KUKA KRL data list: Glode_HanGao.dat

&ACCESS RVO1
&REL 298
&PARAM EDITMASK = *
&PARAM TEMPLATE = C:\KRC\Roboter\Template\vorgabe
&PARAM DISKPATH = KRC:\R1\Program\HK
DEFDAT  glode_hangao PUBLIC




;--------DECL_Enum---------------
GLOBAL ENUM Sink_Type_Enum UpDown_One,LeftRight_One,LeftRight_Two,Null
GLOBAL ENUM Area_Enum L0,C45,L90,C135,L180,C225,L270,C315,N45,N135,N225,N315
GLOBAL ENUM Pos_Type_Enum C_LIN_POS,C_CIR_POS,L_LIN_POS
GLOBAL ENUM Work_Area_Enum A0,A90,A270
GLOBAL ENUM Vision_Model_Enum Calibration,Find_Model
;----------------------------------
;---DECL-STRUC-------------------------


GLOBAL STRUC Surround_Welding_Type BOOL Write_Status,REAL Sink_Size_Long,REAL Sink_Size_Width,REAL Sink_Size_R,REAL Sink_Size_Short_Side,REAL Sink_Size_Short_OnePos,REAL Sink_Size_Short_TwoPos,REAL Sink_Size_Pots_Thick,REAL Sink_Size_Panel_Thick,INT Sink_Model,REAL Sink_Size_Left_Distance,REAL Sink_Size_Down_Distance,Sink_Type_Enum Sink_Type
GLOBAL STRUC LSC_TOOL_TYP INT LSR_MAX_PWR,INT LSR_MIN_PWR,INT LSR_Prg,REAL SNSR_Prg,INT SNSR_State,REAL GAS_Pressure,INT LSR_Dly,INT GAS_Pre_Flow,INT GAS_Post_Flow
GLOBAL STRUC Offset_POS REAL X,REAL Y,REAL Z,REAL A,REAL B,REAL C
GLOBAL STRUC Offset_CIR REAL C_X,REAL C_Y,REAL C_Z,REAL C_A,REAL C_B,REAL C_C
GLOBAL STRUC Calculate_Lin_Const REAL A,REAL B,REAL C
GLOBAL STRUC Calibration_Sink_TYP REAL Long,REAL Width




GLOBAL STRUC Surr_Welding_Craft_Type CHAR Welding_Name[20],E6POS Welding_Pos,REAL Welding_Power,REAL Welding_Speed,REAL Welding_Angle,INT Welding_CDIS,INT Welding_ACC,Offset_POS Welding_Offset,Offset_CIR Welding_Offset_CIR





;-------------------------------------


;----------DECL_Value----------------------
DECL GLOBAL Surround_Welding_Type SW_DEFAULT={Sink_Size_Long 50.0000,Sink_Size_Width 345.000,Sink_Size_R 10.0000,Sink_Size_Pots_Thick 0.750000,Sink_Size_Panel_Thick 2.85000,Sink_Model 952154,Sink_Type #UpDown_One}
DECL GLOBAL LSC_TOOL_TYP LTDEFAULT={LSR_MAX_PWR 500,LSR_MIN_PWR 50,LSR_Prg 1,SNSR_Prg 1.00000,SNSR_State 0,GAS_Pressure 1.00000,LSR_Dly 100,GAS_Pre_Flow 0,GAS_Post_Flow 0}
DECL GLOBAL Offset_POS FFDEFAULT={X 0.0,Y 0.0,Z 0.0,A 0.0,B 0.0,C 0.0}
DECL GLOBAL Offset_CIR FCDEFAULT={C_X 0.0,C_Y 0.0,C_Z 0.0,C_A 0.0,C_B 0.0,C_C 0.0}
DECL GLOBAL E6POS PODEFAULT={X 0.0,Y 0.0,Z 0.0,A 0.0,B 0.0,C 0.0}


DECL GLOBAL Surround_Welding_Type Camera_Calibration_Data={Sink_Size_Long 632.000,Sink_Size_Width 352.000,Sink_Size_R 10.0000,Sink_Size_Short_Side 23.0000,Sink_Size_Short_OnePos 36.0000,Sink_Size_Short_TwoPos 328.000,Sink_Size_Pots_Thick 0.750000,Sink_Size_Panel_Thick 0.0,Sink_Model 952154,Sink_Size_Left_Distance 24.0000,Sink_Size_Down_Distance 24.0000,Sink_Type #LeftRight_One}

DECL GLOBAL E6POS N1_Cam_45_POS={X 1765.00,Y -1.00106740E-34,Z 1784.00,A 0.0,B 90.0000,C 3.24968513E-36}
DECL GLOBAL E6POS N1_Cam_135_POS={X 1765.00,Y -9.34353299E-23,Z 1784.00,A 0.0,B 90.0000,C 3.03311614E-24}
DECL GLOBAL E6POS N1_Cam_225_POS={X 1765.00,Y 5.47478833E-11,Z 1784.00,A 0.0,B 90.0000,C -6.59667199E-13}
DECL GLOBAL E6POS N1_Cam_315_POS={X 0.0,Y 0.0,A 0.0,B 0.0,C 0.0}

DECL GLOBAL E6POS N2_Cam_45_POS={X 293.122131,Y 89.9176636,Z -80.0293961,A 0.441927105,B -0.0416148715,C -0.0704164580,S 'B0010',T 'B1010',E1 0.0,E2 0.0,E3 0.0,E4 0.0,E5 0.0,E6 0.0}
DECL GLOBAL E6POS N2_Cam_135_POS={X -42.3839874,Y 91.8151550,Z -80.0254822,A 0.441927105,B -0.0416148864,C -0.0704164430,S 'B0010',T 'B1010',E1 0.0,E2 0.0,E3 0.0,E4 0.0,E5 0.0,E6 0.0}
DECL GLOBAL E6POS N2_Cam_225_POS={X -39.7999954,Y 716.082336,Z -80.0293350,A 0.441926539,B -0.0416153781,C -0.0704161152,S 'B0010',T 'B00101011',E1 0.0,E2 0.0,E3 0.0,E4 0.0,E5 0.0,E6 0.0}
DECL GLOBAL E6POS N2_Cam_315_POS={X 294.984924,Y 714.198059,Z -80.0293350,A 0.441925645,B -0.0416159667,C -0.0704158247,S 'B0010',T 'B00101011',E1 0.0,E2 0.0,E3 0.0,E4 0.0,E5 0.0,E6 0.0}

DECL GLOBAL E6POS N45_OFFSET_POS={X 375.675,Y 23.4770,Z 0.0,A 0.0,B 0.0,C 0.0}
DECL GLOBAL E6POS N135_OFFSET_POS={X 24.0190,Y 23.1910,Z 0.0,A 0.0,B 0.0,C 0.0}
DECL GLOBAL E6POS N225_OFFSET_POS={X 23.4020,Y 725.222,Z 0.0,A 0.0,B 0.0,C 0.0}
DECL GLOBAL E6POS N315_OFFSET_POS={X 375.730,Y 725.747,Z 0.0,A 0.0,B 0.0,C 0.0}

DECL GLOBAL E6POS N45_CIR_POS={X 372.590,Y 27.2660,Z 0.0,A 0.0,B 0.0,C 0.0}
DECL GLOBAL E6POS N135_CIR_POS={X 27.7730,Y 26.2530,Z 0.0,A 0.0,B 0.0,C 0.0}
DECL GLOBAL E6POS N225_CIR_POS={X 27.3020,Y 722.048,Z 0.0,A 0.0,B 0.0,C 0.0}
DECL GLOBAL E6POS N315_CIR_POS={X 372.023,Y 722.369,Z 0.0,A 0.0,B 0.0,C 0.0}

DECL GLOBAL E6POS D45_Start_POS={X 364.343,Y -0.734000,Z 0.0,A 0.0,B 0.0,C 0.0}
DECL GLOBAL E6POS D45_End_POS={X 364.315,Y 23.5880,Z 0.0,A 0.0,B 0.0,C 0.0}
DECL GLOBAL E6POS D135_Start_POS={X 37.1160,Y -1.02700,Z 0.0,A 0.0,B 0.0,C 0.0}
DECL GLOBAL E6POS D135_End_POS={X 37.2780,Y 23.2150,Z 0.0,A 0.0,B 0.0,C 0.0}
DECL GLOBAL E6POS D225_Start_POS={X 36.7810,Y 749.275,Z 0.0,A 0.0,B 0.0,C 0.0}
DECL GLOBAL E6POS D225_End_POS={X 36.9310,Y 725.260,Z 0.0,A 0.0,B 0.0,C 0.0}
DECL GLOBAL E6POS D315_Start_POS={X 364.063,Y 750.089,Z 0.0,A 0.0,B 0.0,C 0.0}
DECL GLOBAL E6POS D315_End_POS={X 364.380,Y 725.694,Z 0.0,A 0.0,B 0.0,C 0.0}


DECL GLOBAL Surr_Welding_Craft_Type L0_Welding_Craft[2,10]
L0_Welding_Craft[1,1]={Welding_Name[] "S2",Welding_Pos {X 120.000,Y 38.0000,Z 0.0,A 0.0,B 20.0000,C 0.0},Welding_Power 80.0000,Welding_Speed 0.0400000,Welding_Angle 20.0000,Welding_CDIS 5,Welding_ACC 100,Welding_Offset {X 0.0,Y 0.0,Z 0.0}}
L0_Welding_Craft[1,2]={Welding_Name[] "L0_S2",Welding_Pos {X 376.000,Y 584.800,Z 0.0,A 0.0,B 20.0000,C 0.0},Welding_Power 80.0000,Welding_Speed 0.0400000,Welding_Angle 20.0000,Welding_CDIS 5,Welding_ACC 100,Welding_Offset {X 0.0,Y 0.0,Z 0.0}}
L0_Welding_Craft[1,3]={Welding_Name[] "L0_S3",Welding_Pos {X 376.000,Y 340.000,Z 0.0,A 0.0,B 20.0000,C 0.0},Welding_Power 80.0000,Welding_Speed 0.0400000,Welding_Angle 20.0000,Welding_CDIS 5,Welding_ACC 100,Welding_Offset {X 0.0,Y 0.0,Z 0.0}}
L0_Welding_Craft[1,4]={Welding_Name[] "L0_S4",Welding_Pos {X 376.000,Y 64.6000061,Z 0.0,A 0.0,B 20.0000,C 0.0},Welding_Power 80.0000,Welding_Speed 0.0400000,Welding_Angle 20.0000,Welding_CDIS 5,Welding_ACC 100,Welding_Offset {X 0.0,Y 0.0,Z 0.0}}
L0_Welding_Craft[1,5]={Welding_Name[] "S1",Welding_Pos {X 400.000,Y 86.0000153,Z -3.00000,A 0.0,B 23.0000,C 0.0},Welding_Power 80.0000,Welding_Speed 0.0400000,Welding_Angle 20.0000,Welding_CDIS 5,Welding_ACC 100,Welding_Offset {X 0.0,Y 0.0,Z 0.0}}
L0_Welding_Craft[1,6]={Welding_Name[] "S6",Welding_Pos {X 533.000,Y 463.600037,Z -2.05000,A 0.0,B -23.0000,C 0.0},Welding_Power 80.0000,Welding_Speed 0.0400000,Welding_Angle 20.0000,Welding_CDIS 5,Welding_ACC 100,Welding_Offset {X 0.0,Y 0.0,Z 0.0}}
L0_Welding_Craft[1,7]={Welding_Name[] "S7",Welding_Pos {X 533.000,Y 463.600037,Z -2.05000,A 0.0,B -23.0000,C 0.0},Welding_Power 80.0000,Welding_Speed 0.0400000,Welding_Angle 20.0000,Welding_CDIS 5,Welding_ACC 100,Welding_Offset {X 0.0,Y 0.0,Z 0.0}}
L0_Welding_Craft[1,8]={Welding_Name[] "S8",Welding_Pos {X 533.000,Y 463.600037,Z -2.05000,A 0.0,B -23.0000,C 0.0},Welding_Power 80.0000,Welding_Speed 0.0400000,Welding_Angle 20.0000,Welding_CDIS 5,Welding_ACC 100,Welding_Offset {X 0.0,Y 0.0,Z 0.0}}
L0_Welding_Craft[1,9]={Welding_Name[] "S9",Welding_Pos {X 533.000,Y 463.600037,Z -2.05000,A 0.0,B -23.0000,C 0.0},Welding_Power 80.0000,Welding_Speed 0.0400000,Welding_Angle 20.0000,Welding_CDIS 5,Welding_ACC 100,Welding_Offset {X 0.0,Y 0.0,Z 0.0}}
L0_Welding_Craft[1,10]={Welding_Name[] "S10",Welding_Pos {X 533.000,Y 338.000,Z -2.05000,A 0.0,B -23.0000,C 0.0},Welding_Power 80.0000,Welding_Speed 0.0400000,Welding_Angle 20.0000,Welding_CDIS 5,Welding_ACC 100,Welding_Offset {X 0.0,Y 0.0,Z 0.0}}
L0_Welding_Craft[2,1]={Welding_Name[] "L0_S1",Welding_Pos {X 375.681122,Y 101.703979,Z 0.0,A 0.0,B 20.0000,C 0.0},Welding_Power 80.0000,Welding_Speed 0.300000,Welding_Angle 20.0000,Welding_CDIS 5,Welding_ACC 100,Welding_Offset {X 0.0,Y 0.0,Z 0.0}}
L0_Welding_Craft[2,2]={Welding_Name[] "L0_S2",Welding_Pos {X 375.566071,Y 647.351257,Z 0.0,A 0.0,B 20.0000,C 0.0},Welding_Power 80.0000,Welding_Speed 0.0320000,Welding_Angle 20.0000,Welding_CDIS 5,Welding_ACC 100,Welding_Offset {X 0.0,Y -1.50000,Z 0.0}}
L0_Welding_Craft[2,3]={Welding_Name[] "L0_S3",Welding_Pos {X 375.650,Y 374.428497,Z 0.0,A 0.0,B 20.0000,C 0.0},Welding_Power 80.0000,Welding_Speed 0.0320000,Welding_Angle 20.0000,Welding_CDIS 5,Welding_ACC 100,Welding_Offset {X 0.0,Y -1.80000,Z 0.0}}
L0_Welding_Craft[2,4]={Welding_Name[] "L0_S4",Welding_Pos {X 375.744415,Y 67.3903809,Z 0.0,A 0.0,B 20.0000,C 0.0},Welding_Power 80.0000,Welding_Speed 0.0340000,Welding_Angle 20.0000,Welding_CDIS 5,Welding_ACC 100,Welding_Offset {X 0.0,Y -1.00000,Z 0.0}}
L0_Welding_Craft[2,5]={Welding_Name[] "S1",Welding_Pos {X 400.000,Y 86.0000153,Z -3.00000,A 0.0,B 23.0000,C 0.0},Welding_Power 80.0000,Welding_Speed 0.0400000,Welding_Angle 20.0000,Welding_CDIS 5,Welding_ACC 100,Welding_Offset {X 0.0,Y 0.0,Z 0.0}}
L0_Welding_Craft[2,6]={Welding_Name[] "S6",Welding_Pos {X 533.000,Y 463.600037,Z -2.05000,A 0.0,B -23.0000,C 0.0},Welding_Power 80.0000,Welding_Speed 0.0400000,Welding_Angle 20.0000,Welding_CDIS 5,Welding_ACC 100,Welding_Offset {X 0.0,Y 0.0,Z 0.0}}
L0_Welding_Craft[2,7]={Welding_Name[] "S7",Welding_Pos {X 533.000,Y 463.600037,Z -2.05000,A 0.0,B -23.0000,C 0.0},Welding_Power 80.0000,Welding_Speed 0.0400000,Welding_Angle 20.0000,Welding_CDIS 5,Welding_ACC 100,Welding_Offset {X 0.0,Y 0.0,Z 0.0}}
L0_Welding_Craft[2,8]={Welding_Name[] "S8",Welding_Pos {X 533.000,Y 463.600037,Z -2.05000,A 0.0,B -23.0000,C 0.0},Welding_Power 80.0000,Welding_Speed 0.0400000,Welding_Angle 20.0000,Welding_CDIS 5,Welding_ACC 100,Welding_Offset {X 0.0,Y 0.0,Z 0.0}}
L0_Welding_Craft[2,9]={Welding_Name[] "S9",Welding_Pos {X 533.000,Y 463.600037,Z -2.05000,A 0.0,B -23.0000,C 0.0},Welding_Power 80.0000,Welding_Speed 0.0400000,Welding_Angle 20.0000,Welding_CDIS 5,Welding_ACC 100,Welding_Offset {X 0.0,Y 0.0,Z 0.0}}
L0_Welding_Craft[2,10]={Welding_Name[] "S10",Welding_Pos {X 533.000,Y 338.000,Z -2.05000,A 0.0,B -23.0000,C 0.0},Welding_Power 80.0000,Welding_Speed 0.0400000,Welding_Angle 20.0000,Welding_CDIS 5,Welding_ACC 100,Welding_Offset {X 0.0,Y 0.0,Z 0.0}}



DECL GLOBAL Surr_Welding_Craft_Type C45_Welding_Craft[2,3]
C45_Welding_Craft[1,1]={Welding_Name[] "S3",Welding_Pos {X 120.000,Y 30.0000,Z 0.0,A 0.0,B 20.0000,C 0.0},Welding_Power 80.0000,Welding_Speed 0.0400000,Welding_Angle 20.0000,Welding_CDIS 5,Welding_ACC 100,Welding_Offset {X 0.0,Y 0.0,Z 0.0}}
C45_Welding_Craft[1,2]={Welding_Name[] "PM2",Welding_Pos {X 117.070,Y 22.9300,Z 0.0,A 0.0,B 0.0,C 0.0},Welding_Power 80.0000,Welding_Speed 0.0400000,Welding_Angle 20.0000,Welding_CDIS 5,Welding_ACC 100,Welding_Offset {X 0.0,Y 0.0,Z 0.0},Welding_Offset_CIR {C_X 0.0,C_Y 0.0,C_Z 0.0}}
C45_Welding_Craft[1,3]={Welding_Name[] "PE2",Welding_Pos {X 110.000,Y 20.0000,Z 0.0,A 0.0,B 0.0,C 20.0000},Welding_Power 80.0000,Welding_Speed 0.0400000,Welding_Angle 20.0000,Welding_CDIS 5,Welding_ACC 100,Welding_Offset {X 0.0,Y 0.0,Z 0.0}}
C45_Welding_Craft[2,1]={Welding_Name[] "C45_S1",Welding_Pos {X 375.754913,Y 33.2750244,Z 0.0,A 0.0,B 20.0000,C 0.0},Welding_Power 80.0000,Welding_Speed 0.0300000,Welding_Angle 20.0000,Welding_CDIS 5,Welding_ACC 100,Welding_Offset {X 0.0,Y 0.0,Z 0.0}}
C45_Welding_Craft[2,2]={Welding_Name[] "PM3",Welding_Pos {X 372.649,Y 27.0560,Z 0.0,A 0.0,B 0.0,C 0.0},Welding_Power 80.0000,Welding_Speed 0.0400000,Welding_Angle 20.0000,Welding_CDIS 5,Welding_ACC 100,Welding_Offset {X 0.0,Y 0.500000,Z 0.0},Welding_Offset_CIR {C_X 0.0,C_Y 0.0,C_Z 0.0}}
C45_Welding_Craft[2,3]={Welding_Name[] "PE3",Welding_Pos {X 365.758,Y 23.2745743,Z 0.0,A 0.0,B 0.0,C 20.0000},Welding_Power 80.0000,Welding_Speed 0.0120000,Welding_Angle 20.0000,Welding_CDIS 5,Welding_ACC 100,Welding_Offset {X 0.0,Y 0.500000,Z 0.0}}


DECL GLOBAL Surr_Welding_Craft_Type L90_Welding_Craft[2,10]
L90_Welding_Craft[1,1]={Welding_Name[] "S2",Welding_Pos {X 30.0000,Y 20.0000,Z 0.0,A 0.0,B 0.0,C 20.0000},Welding_Power 80.0000,Welding_Speed 0.0400000,Welding_Angle 20.0000,Welding_CDIS 5,Welding_ACC 100,Welding_Offset {X 0.0,Y 0.0,Z 0.0}}
L90_Welding_Craft[1,2]={Welding_Name[] "L90_S2",Welding_Pos {X 200.000,Y 24.0000,Z 0.0,A 0.0,B 0.0,C 20.0000},Welding_Power 80.0000,Welding_Speed 0.0400000,Welding_Angle 20.0000,Welding_CDIS 5,Welding_ACC 100,Welding_Offset {X 0.0,Y 0.0,Z 0.0}}
L90_Welding_Craft[1,3]={Welding_Name[] "L90_S3",Welding_Pos {X 67.2000122,Y 24.0000,Z 0.0,A 0.0,B 0.0,C 20.0000},Welding_Power 80.0000,Welding_Speed 0.0400000,Welding_Angle 20.0000,Welding_CDIS 5,Welding_ACC 100,Welding_Offset {X 0.0,Y 0.0,Z 0.0}}
L90_Welding_Craft[1,4]={Welding_Name[] "S4",Welding_Pos {X 400.000,Y 86.0000153,Z -3.00000,A 0.0,B 23.0000,C 0.0},Welding_Power 80.0000,Welding_Speed 0.0400000,Welding_Angle 20.0000,Welding_CDIS 5,Welding_ACC 100,Welding_Offset {X 0.0,Y 0.0,Z 0.0}}
L90_Welding_Craft[1,5]={Welding_Name[] "S5",Welding_Pos {X 371.000,Y 0.0,Z -3.00000,A 0.0,B 0.0,C 23.0000},Welding_Power 80.0000,Welding_Speed 0.0400000,Welding_Angle 20.0000,Welding_CDIS 5,Welding_ACC 100,Welding_Offset {X 0.0,Y 0.0,Z 0.0}}
L90_Welding_Craft[1,6]={Welding_Name[] "S6",Welding_Pos {X 533.000,Y 463.600037,Z -2.05000,A 0.0,B -23.0000,C 0.0},Welding_Power 80.0000,Welding_Speed 0.0400000,Welding_Angle 20.0000,Welding_CDIS 5,Welding_ACC 100,Welding_Offset {X 0.0,Y 0.0,Z 0.0}}
L90_Welding_Craft[1,7]={Welding_Name[] "S7",Welding_Pos {X 533.000,Y 463.600037,Z -2.05000,A 0.0,B -23.0000,C 0.0},Welding_Power 80.0000,Welding_Speed 0.0400000,Welding_Angle 20.0000,Welding_CDIS 5,Welding_ACC 100,Welding_Offset {X 0.0,Y 0.0,Z 0.0}}
L90_Welding_Craft[1,8]={Welding_Name[] "S8",Welding_Pos {X 533.000,Y 463.600037,Z -2.05000,A 0.0,B -23.0000,C 0.0},Welding_Power 80.0000,Welding_Speed 0.0400000,Welding_Angle 20.0000,Welding_CDIS 5,Welding_ACC 100,Welding_Offset {X 0.0,Y 0.0,Z 0.0}}
L90_Welding_Craft[1,9]={Welding_Name[] "S9",Welding_Pos {X 533.000,Y 463.600037,Z -2.05000,A 0.0,B -23.0000,C 0.0},Welding_Power 80.0000,Welding_Speed 0.0400000,Welding_Angle 20.0000,Welding_CDIS 5,Welding_ACC 100,Welding_Offset {X 0.0,Y 0.0,Z 0.0}}
L90_Welding_Craft[1,10]={Welding_Name[] "S10",Welding_Pos {X 533.000,Y 338.000,Z -2.05000,A 0.0,B -23.0000,C 0.0},Welding_Power 80.0000,Welding_Speed 0.0400000,Welding_Angle 20.0000,Welding_CDIS 5,Welding_ACC 100,Welding_Offset {X 0.0,Y 0.0,Z 0.0}}
L90_Welding_Craft[2,1]={Welding_Name[] "L90_S1",Welding_Pos {X 332.548584,Y 23.2731590,Z 0.0,A 0.0,B 0.0,C 20.0000},Welding_Power 80.0000,Welding_Speed 0.0320000,Welding_Angle 20.0000,Welding_CDIS 5,Welding_ACC 100,Welding_Offset {X 0.0,Y 0.800000,Z 0.0}}
L90_Welding_Craft[2,2]={Welding_Name[] "L90_S2",Welding_Pos {X 199.711,Y 23.2675,Z 0.0,A 0.0,B 0.0,C 20.0000},Welding_Power 80.0000,Welding_Speed 0.0320000,Welding_Angle 20.0000,Welding_CDIS 5,Welding_ACC 100,Welding_Offset {X 0.0,Y 0.800000,Z 0.0}}
L90_Welding_Craft[2,3]={Welding_Name[] "L90_S3",Welding_Pos {X 66.8734131,Y 23.2618408,Z 0.0,A 0.0,B 0.0,C 20.0000},Welding_Power 80.0000,Welding_Speed 0.0320000,Welding_Angle 20.0000,Welding_CDIS 5,Welding_ACC 100,Welding_Offset {X 0.0,Y 0.800000,Z 0.0}}
L90_Welding_Craft[2,4]={Welding_Name[] "S4",Welding_Pos {X 400.000,Y 86.0000153,Z -3.00000,A 0.0,B 23.0000,C 0.0},Welding_Power 80.0000,Welding_Speed 0.0400000,Welding_Angle 20.0000,Welding_CDIS 5,Welding_ACC 100,Welding_Offset {X 0.0,Y 0.0,Z 0.0}}
L90_Welding_Craft[2,5]={Welding_Name[] "S5",Welding_Pos {X 371.000,Y 0.0,Z -3.00000,A 0.0,B 0.0,C 23.0000},Welding_Power 80.0000,Welding_Speed 0.0400000,Welding_Angle 20.0000,Welding_CDIS 5,Welding_ACC 100,Welding_Offset {X 0.0,Y 0.0,Z 0.0}}
L90_Welding_Craft[2,6]={Welding_Name[] "S6",Welding_Pos {X 533.000,Y 463.600037,Z -2.05000,A 0.0,B -23.0000,C 0.0},Welding_Power 80.0000,Welding_Speed 0.0400000,Welding_Angle 20.0000,Welding_CDIS 5,Welding_ACC 100,Welding_Offset {X 0.0,Y 0.0,Z 0.0}}
L90_Welding_Craft[2,7]={Welding_Name[] "S7",Welding_Pos {X 533.000,Y 463.600037,Z -2.05000,A 0.0,B -23.0000,C 0.0},Welding_Power 80.0000,Welding_Speed 0.0400000,Welding_Angle 20.0000,Welding_CDIS 5,Welding_ACC 100,Welding_Offset {X 0.0,Y 0.0,Z 0.0}}
L90_Welding_Craft[2,8]={Welding_Name[] "S8",Welding_Pos {X 533.000,Y 463.600037,Z -2.05000,A 0.0,B -23.0000,C 0.0},Welding_Power 80.0000,Welding_Speed 0.0400000,Welding_Angle 20.0000,Welding_CDIS 5,Welding_ACC 100,Welding_Offset {X 0.0,Y 0.0,Z 0.0}}
L90_Welding_Craft[2,9]={Welding_Name[] "S9",Welding_Pos {X 533.000,Y 463.600037,Z -2.05000,A 0.0,B -23.0000,C 0.0},Welding_Power 80.0000,Welding_Speed 0.0400000,Welding_Angle 20.0000,Welding_CDIS 5,Welding_ACC 100,Welding_Offset {X 0.0,Y 0.0,Z 0.0}}
L90_Welding_Craft[2,10]={Welding_Name[] "S10",Welding_Pos {X 533.000,Y 338.000,Z -2.05000,A 0.0,B -23.0000,C 0.0},Welding_Power 80.0000,Welding_Speed 0.0400000,Welding_Angle 20.0000,Welding_CDIS 5,Welding_ACC 100,Welding_Offset {X 0.0,Y 0.0,Z 0.0}}

DECL GLOBAL Surr_Welding_Craft_Type C135_Welding_Craft[2,3]
C135_Welding_Craft[1,1]={Welding_Name[] "S3",Welding_Pos {X 30.0000,Y 20.0000,Z 0.0,A 0.0,B 0.0,C 20.0000},Welding_Power 80.0000,Welding_Speed 0.0400000,Welding_Angle 20.0000,Welding_CDIS 5,Welding_ACC 100,Welding_Offset {X 0.0,Y 0.0,Z 0.0}}
C135_Welding_Craft[1,2]={Welding_Name[] "PM3",Welding_Pos {X 22.9300,Y 22.9300,Z 0.0,A 0.0,B 0.0,C 0.0},Welding_Power 80.0000,Welding_Speed 0.0400000,Welding_Angle -20.0000,Welding_CDIS 5,Welding_ACC 100,Welding_Offset {X 0.0,Y 0.0,Z 0.0},Welding_Offset_CIR {C_X 0.0,C_Y 0.0,C_Z 0.0}}
C135_Welding_Craft[1,3]={Welding_Name[] "PE3",Welding_Pos {X 20.0000,Y 30.0000,Z 0.0,A 0.0,B -20.0000,C 0.0},Welding_Power 80.0000,Welding_Speed 0.0400000,Welding_Angle -20.0000,Welding_CDIS 5,Welding_ACC 100,Welding_Offset {X 0.0,Y 0.0,Z 0.0}}
C135_Welding_Craft[2,1]={Welding_Name[] "C135_S1",Welding_Pos {X 33.6640,Y 23.2604256,Z 0.0,A 0.0,B 0.0,C 20.0000},Welding_Power 80.0000,Welding_Speed 0.0300000,Welding_Angle 20.0000,Welding_CDIS 5,Welding_ACC 100,Welding_Offset {X 0.0,Y 0.500000,Z 0.0}}
C135_Welding_Craft[2,2]={Welding_Name[] "PM4",Welding_Pos {X 27.4390,Y 26.3430,Z 0.0,A 0.0,B 0.0,C 0.0},Welding_Power 80.0000,Welding_Speed 0.0400000,Welding_Angle -20.0000,Welding_CDIS 5,Welding_ACC 100,Welding_Offset {X 0.0,Y 0.0,Z 0.0},Welding_Offset_CIR {C_X 0.0,C_Y 0.0,C_Z 0.0}}
C135_Welding_Craft[2,3]={Welding_Name[] "PE4",Welding_Pos {X 23.6575489,Y 33.2600,Z 0.0,A 0.0,B -20.0000,C 0.0},Welding_Power 80.0000,Welding_Speed 0.0150000,Welding_Angle -20.0000,Welding_CDIS 5,Welding_ACC 100,Welding_Offset {X 0.0,Y 0.500000,Z 0.0}}

DECL GLOBAL Surr_Welding_Craft_Type L180_Welding_Craft[2,10]
L180_Welding_Craft[1,1]={Welding_Name[] "S2",Welding_Pos {X 20.0000,Y 30.0000,Z 0.0,A 0.0,B -20.0000,C 0.0},Welding_Power 80.0000,Welding_Speed 0.0400000,Welding_Angle -20.0000,Welding_CDIS 5,Welding_ACC 100,Welding_Offset {X 0.0,Y 0.0,Z 0.0}}
L180_Welding_Craft[1,2]={Welding_Name[] "L180_S2",Welding_Pos {X 24.0000,Y 340.000,Z 0.0,A 0.0,B -20.0000,C 0.0},Welding_Power 80.0000,Welding_Speed 0.0400000,Welding_Angle -20.0000,Welding_CDIS 5,Welding_ACC 100,Welding_Offset {X 0.0,Y 0.0,Z 0.0}}
L180_Welding_Craft[1,3]={Welding_Name[] "L180_S3",Welding_Pos {X 24.0000,Y 615.399963,Z 0.0,A 0.0,B -20.0000,C 0.0},Welding_Power 80.0000,Welding_Speed 0.0400000,Welding_Angle -20.0000,Welding_CDIS 5,Welding_ACC 100,Welding_Offset {X 0.0,Y 0.0,Z 0.0}}
L180_Welding_Craft[1,4]={Welding_Name[] "S4",Welding_Pos {X 400.000,Y 86.0000153,Z -3.00000,A 0.0,B 23.0000,C 0.0},Welding_Power 80.0000,Welding_Speed 0.0400000,Welding_Angle -20.0000,Welding_CDIS 5,Welding_ACC 100,Welding_Offset {X 0.0,Y 0.0,Z 0.0}}
L180_Welding_Craft[1,5]={Welding_Name[] "S5",Welding_Pos {X 0.0,Y 371.000,Z -3.00000,A 0.0,B -23.0000,C 0.0},Welding_Power 80.0000,Welding_Speed 0.0400000,Welding_Angle -20.0000,Welding_CDIS 5,Welding_ACC 100,Welding_Offset {X 0.0,Y 0.0,Z 0.0}}
L180_Welding_Craft[1,6]={Welding_Name[] "S6",Welding_Pos {X 533.000,Y 463.600037,Z -2.05000,A 0.0,B -23.0000,C 0.0},Welding_Power 80.0000,Welding_Speed 0.0400000,Welding_Angle -20.0000,Welding_CDIS 5,Welding_ACC 100,Welding_Offset {X 0.0,Y 0.0,Z 0.0}}
L180_Welding_Craft[1,7]={Welding_Name[] "S7",Welding_Pos {X 533.000,Y 463.600037,Z -2.05000,A 0.0,B -23.0000,C 0.0},Welding_Power 80.0000,Welding_Speed 0.0400000,Welding_Angle -20.0000,Welding_CDIS 5,Welding_ACC 100,Welding_Offset {X 0.0,Y 0.0,Z 0.0}}
L180_Welding_Craft[1,8]={Welding_Name[] "S8",Welding_Pos {X 533.000,Y 463.600037,Z -2.05000,A 0.0,B -23.0000,C 0.0},Welding_Power 80.0000,Welding_Speed 0.0400000,Welding_Angle -20.0000,Welding_CDIS 5,Welding_ACC 100,Welding_Offset {X 0.0,Y 0.0,Z 0.0}}
L180_Welding_Craft[1,9]={Welding_Name[] "S9",Welding_Pos {X 533.000,Y 463.600037,Z -2.05000,A 0.0,B -23.0000,C 0.0},Welding_Power 80.0000,Welding_Speed 0.0400000,Welding_Angle -20.0000,Welding_CDIS 5,Welding_ACC 100,Welding_Offset {X 0.0,Y 0.0,Z 0.0}}
L180_Welding_Craft[1,10]={Welding_Name[] "S10",Welding_Pos {X 533.000,Y 338.000,Z -2.05000,A 0.0,B -23.0000,C 0.0},Welding_Power 80.0000,Welding_Speed 0.0400000,Welding_Angle -20.0000,Welding_CDIS 5,Welding_ACC 100,Welding_Offset {X 0.0,Y 0.0,Z 0.0}}
L180_Welding_Craft[2,1]={Welding_Name[] "L180_S1",Welding_Pos {X 23.6135387,Y 101.477905,Z 0.0,A 0.0,B -20.0000,C 0.0},Welding_Power 80.0000,Welding_Speed 0.0320000,Welding_Angle -20.0000,Welding_CDIS 5,Welding_ACC 100,Welding_Offset {X 0.0,Y 0.0,Z 0.0}}
L180_Welding_Craft[2,2]={Welding_Name[] "L180_S2",Welding_Pos {X 23.4375,Y 374.349518,Z 0.0,A 0.0,B -20.0000,C 0.0},Welding_Power 80.0000,Welding_Speed 0.0320000,Welding_Angle -20.0000,Welding_CDIS 5,Welding_ACC 100,Welding_Offset {X 0.0,Y 0.0,Z 0.0}}
L180_Welding_Craft[2,3]={Welding_Name[] "L180_S3",Welding_Pos {X 23.2394562,Y 681.330078,Z 0.0,A 0.0,B -20.0000,C 0.0},Welding_Power 80.0000,Welding_Speed 0.0320000,Welding_Angle -20.0000,Welding_CDIS 5,Welding_ACC 100,Welding_Offset {X 0.200000,Y 0.0,Z 0.0}}
L180_Welding_Craft[2,4]={Welding_Name[] "S4",Welding_Pos {X 400.000,Y 86.0000153,Z -3.00000,A 0.0,B 23.0000,C 0.0},Welding_Power 80.0000,Welding_Speed 0.0400000,Welding_Angle -20.0000,Welding_CDIS 5,Welding_ACC 100,Welding_Offset {X 0.0,Y 0.0,Z 0.0}}
L180_Welding_Craft[2,5]={Welding_Name[] "S5",Welding_Pos {X 0.0,Y 371.000,Z -3.00000,A 0.0,B -23.0000,C 0.0},Welding_Power 80.0000,Welding_Speed 0.0400000,Welding_Angle -20.0000,Welding_CDIS 5,Welding_ACC 100,Welding_Offset {X 0.0,Y 0.0,Z 0.0}}
L180_Welding_Craft[2,6]={Welding_Name[] "S6",Welding_Pos {X 533.000,Y 463.600037,Z -2.05000,A 0.0,B -23.0000,C 0.0},Welding_Power 80.0000,Welding_Speed 0.0400000,Welding_Angle -20.0000,Welding_CDIS 5,Welding_ACC 100,Welding_Offset {X 0.0,Y 0.0,Z 0.0}}
L180_Welding_Craft[2,7]={Welding_Name[] "S7",Welding_Pos {X 533.000,Y 463.600037,Z -2.05000,A 0.0,B -23.0000,C 0.0},Welding_Power 80.0000,Welding_Speed 0.0400000,Welding_Angle -20.0000,Welding_CDIS 5,Welding_ACC 100,Welding_Offset {X 0.0,Y 0.0,Z 0.0}}
L180_Welding_Craft[2,8]={Welding_Name[] "S8",Welding_Pos {X 533.000,Y 463.600037,Z -2.05000,A 0.0,B -23.0000,C 0.0},Welding_Power 80.0000,Welding_Speed 0.0400000,Welding_Angle -20.0000,Welding_CDIS 5,Welding_ACC 100,Welding_Offset {X 0.0,Y 0.0,Z 0.0}}
L180_Welding_Craft[2,9]={Welding_Name[] "S9",Welding_Pos {X 533.000,Y 463.600037,Z -2.05000,A 0.0,B -23.0000,C 0.0},Welding_Power 80.0000,Welding_Speed 0.0400000,Welding_Angle -20.0000,Welding_CDIS 5,Welding_ACC 100,Welding_Offset {X 0.0,Y 0.0,Z 0.0}}
L180_Welding_Craft[2,10]={Welding_Name[] "S10",Welding_Pos {X 533.000,Y 338.000,Z -2.05000,A 0.0,B -23.0000,C 0.0},Welding_Power 80.0000,Welding_Speed 0.0400000,Welding_Angle -20.0000,Welding_CDIS 5,Welding_ACC 100,Welding_Offset {X 0.0,Y 0.0,Z 0.0}}

DECL GLOBAL Surr_Welding_Craft_Type C225_Welding_Craft[2,3]
C225_Welding_Craft[1,1]={Welding_Name[] "S3",Welding_Pos {X 20.0000,Y 110.000,Z 0.0,A 0.0,B -20.0000,C 0.0},Welding_Power 80.0000,Welding_Speed 0.0400000,Welding_Angle -20.0000,Welding_CDIS 5,Welding_ACC 100,Welding_Offset {X 0.0,Y 0.0,Z 0.0}}
C225_Welding_Craft[1,2]={Welding_Name[] "PM3",Welding_Pos {X 22.9300,Y 117.070,Z 0.0,A 0.0,B 0.0,C 0.0},Welding_Power 80.0000,Welding_Speed 0.0400000,Welding_Angle -20.0000,Welding_CDIS 5,Welding_ACC 100,Welding_Offset {X 0.0,Y 0.0,Z 0.0},Welding_Offset_CIR {C_X 0.0,C_Y 0.0,C_Z 0.0}}
C225_Welding_Craft[1,3]={Welding_Name[] "PE3",Welding_Pos {X 30.0000,Y 120.000,Z 0.0,A 0.0,B 0.0,C -20.0000},Welding_Power 80.0000,Welding_Speed 0.0400000,Welding_Angle -20.0000,Welding_CDIS 5,Welding_ACC 100,Welding_Offset {X 0.0,Y 0.0,Z 0.0}}
C225_Welding_Craft[2,1]={Welding_Name[] "C225_S1",Welding_Pos {X 23.2174511,Y 715.439,Z 0.0,A 0.0,B -20.0000,C 0.0},Welding_Power 80.0000,Welding_Speed 0.0300000,Welding_Angle -20.0000,Welding_CDIS 5,Welding_ACC 100,Welding_Offset {X 0.300000,Y 0.0,Z 0.0}}
C225_Welding_Craft[2,2]={Welding_Name[] "PM5",Welding_Pos {X 27.1170,Y 722.236,Z 0.0,A 0.0,B 0.0,C 0.0},Welding_Power 80.0000,Welding_Speed 0.0400000,Welding_Angle -20.0000,Welding_CDIS 5,Welding_ACC 100,Welding_Offset {X 0.0,Y 0.0,Z 0.0},Welding_Offset_CIR {C_X 0.0,C_Y 0.0,C_Z 0.0}}
C225_Welding_Craft[2,3]={Welding_Name[] "PE5",Welding_Pos {X 33.2110,Y 725.443054,Z 0.0,A 0.0,B 0.0,C -20.0000},Welding_Power 80.0000,Welding_Speed 0.0150000,Welding_Angle -20.0000,Welding_CDIS 5,Welding_ACC 100,Welding_Offset {X 0.0,Y 0.0,Z 0.0}}

DECL GLOBAL Surr_Welding_Craft_Type L270_Welding_Craft[2,10]
L270_Welding_Craft[1,1]={Welding_Name[] "S2",Welding_Pos {X 110.000,Y 120.000,Z 0.0,A 0.0,B 0.0,C -20.0000},Welding_Power 80.0000,Welding_Speed 0.0400000,Welding_Angle -20.0000,Welding_CDIS 5,Welding_ACC 100,Welding_Offset {X 0.0,Y 0.0,Z 0.0}}
L270_Welding_Craft[1,2]={Welding_Name[] "L270_S2",Welding_Pos {X 200.000,Y 656.000,Z 0.0,A 0.0,B 0.0,C -20.0000},Welding_Power 80.0000,Welding_Speed 0.0400000,Welding_Angle -20.0000,Welding_CDIS 5,Welding_ACC 100,Welding_Offset {X 0.0,Y 0.0,Z 0.0}}
L270_Welding_Craft[1,3]={Welding_Name[] "L270_S3",Welding_Pos {X 349.400,Y 656.000,Z 0.0,A 0.0,B 0.0,C -20.0000},Welding_Power 80.0000,Welding_Speed 0.0400000,Welding_Angle -20.0000,Welding_CDIS 5,Welding_ACC 100,Welding_Offset {X 0.0,Y 0.0,Z 0.0}}
L270_Welding_Craft[1,4]={Welding_Name[] "S4",Welding_Pos {X 400.000,Y 86.0000153,Z -3.00000,A 0.0,B 23.0000,C 0.0},Welding_Power 80.0000,Welding_Speed 0.0400000,Welding_Angle -20.0000,Welding_CDIS 5,Welding_ACC 100,Welding_Offset {X 0.0,Y 0.0,Z 0.0}}
L270_Welding_Craft[1,5]={Welding_Name[] "S12",Welding_Pos {X 28.9999981,Y 400.000,Z -3.00000,A 0.0,B 0.0,C -23.0000},Welding_Power 80.0000,Welding_Speed 0.0400000,Welding_Angle -20.0000,Welding_CDIS 5,Welding_ACC 100,Welding_Offset {X 0.0,Y 0.0,Z 0.0}}
L270_Welding_Craft[1,6]={Welding_Name[] "S6",Welding_Pos {X 533.000,Y 463.600037,Z -2.05000,A 0.0,B -23.0000,C 0.0},Welding_Power 80.0000,Welding_Speed 0.0400000,Welding_Angle -20.0000,Welding_CDIS 5,Welding_ACC 100,Welding_Offset {X 0.0,Y 0.0,Z 0.0}}
L270_Welding_Craft[1,7]={Welding_Name[] "S7",Welding_Pos {X 533.000,Y 463.600037,Z -2.05000,A 0.0,B -23.0000,C 0.0},Welding_Power 80.0000,Welding_Speed 0.0400000,Welding_Angle -20.0000,Welding_CDIS 5,Welding_ACC 100,Welding_Offset {X 0.0,Y 0.0,Z 0.0}}
L270_Welding_Craft[1,8]={Welding_Name[] "S8",Welding_Pos {X 533.000,Y 463.600037,Z -2.05000,A 0.0,B -23.0000,C 0.0},Welding_Power 80.0000,Welding_Speed 0.0400000,Welding_Angle -20.0000,Welding_CDIS 5,Welding_ACC 100,Welding_Offset {X 0.0,Y 0.0,Z 0.0}}
L270_Welding_Craft[1,9]={Welding_Name[] "S9",Welding_Pos {X 533.000,Y 463.600037,Z -2.05000,A 0.0,B -23.0000,C 0.0},Welding_Power 80.0000,Welding_Speed 0.0400000,Welding_Angle -20.0000,Welding_CDIS 5,Welding_ACC 100,Welding_Offset {X 0.0,Y 0.0,Z 0.0}}
L270_Welding_Craft[1,10]={Welding_Name[] "S10",Welding_Pos {X 533.000,Y 338.000,Z -2.05000,A 0.0,B -23.0000,C 0.0},Welding_Power 80.0000,Welding_Speed 0.0400000,Welding_Angle -20.0000,Welding_CDIS 5,Welding_ACC 100,Welding_Offset {X 0.0,Y 0.0,Z 0.0}}
L270_Welding_Craft[2,1]={Welding_Name[] "L270_S1",Welding_Pos {X 66.4440918,Y 725.456543,Z 0.0,A 0.0,B 0.0,C -20.0000},Welding_Power 80.0000,Welding_Speed 0.0320000,Welding_Angle -20.0000,Welding_CDIS 5,Welding_ACC 100,Welding_Offset {X 0.0,Y 0.0,Z 0.0}}
L270_Welding_Craft[2,2]={Welding_Name[] "L270_S2",Welding_Pos {X 199.376495,Y 725.510498,Z 0.0,A 0.0,B 0.0,C -20.0000},Welding_Power 80.0000,Welding_Speed 0.0320000,Welding_Angle -20.0000,Welding_CDIS 5,Welding_ACC 100,Welding_Offset {X 0.0,Y 0.0,Z 0.0}}
L270_Welding_Craft[2,3]={Welding_Name[] "L270_S3",Welding_Pos {X 348.925446,Y 725.571167,Z 0.0,A 0.0,B 0.0,C -20.0000},Welding_Power 80.0000,Welding_Speed 0.0320000,Welding_Angle -20.0000,Welding_CDIS 5,Welding_ACC 100,Welding_Offset {X 0.0,Y 0.0,Z 0.0}}
L270_Welding_Craft[2,4]={Welding_Name[] "S4",Welding_Pos {X 400.000,Y 86.0000153,Z -3.00000,A 0.0,B 23.0000,C 0.0},Welding_Power 80.0000,Welding_Speed 0.0400000,Welding_Angle -20.0000,Welding_CDIS 5,Welding_ACC 100,Welding_Offset {X 0.0,Y 0.0,Z 0.0}}
L270_Welding_Craft[2,5]={Welding_Name[] "S12",Welding_Pos {X 28.9999981,Y 400.000,Z -3.00000,A 0.0,B 0.0,C -23.0000},Welding_Power 80.0000,Welding_Speed 0.0400000,Welding_Angle -20.0000,Welding_CDIS 5,Welding_ACC 100,Welding_Offset {X 0.0,Y 0.0,Z 0.0}}
L270_Welding_Craft[2,6]={Welding_Name[] "S6",Welding_Pos {X 533.000,Y 463.600037,Z -2.05000,A 0.0,B -23.0000,C 0.0},Welding_Power 80.0000,Welding_Speed 0.0400000,Welding_Angle -20.0000,Welding_CDIS 5,Welding_ACC 100,Welding_Offset {X 0.0,Y 0.0,Z 0.0}}
L270_Welding_Craft[2,7]={Welding_Name[] "S7",Welding_Pos {X 533.000,Y 463.600037,Z -2.05000,A 0.0,B -23.0000,C 0.0},Welding_Power 80.0000,Welding_Speed 0.0400000,Welding_Angle -20.0000,Welding_CDIS 5,Welding_ACC 100,Welding_Offset {X 0.0,Y 0.0,Z 0.0}}
L270_Welding_Craft[2,8]={Welding_Name[] "S8",Welding_Pos {X 533.000,Y 463.600037,Z -2.05000,A 0.0,B -23.0000,C 0.0},Welding_Power 80.0000,Welding_Speed 0.0400000,Welding_Angle -20.0000,Welding_CDIS 5,Welding_ACC 100,Welding_Offset {X 0.0,Y 0.0,Z 0.0}}
L270_Welding_Craft[2,9]={Welding_Name[] "S9",Welding_Pos {X 533.000,Y 463.600037,Z -2.05000,A 0.0,B -23.0000,C 0.0},Welding_Power 80.0000,Welding_Speed 0.0400000,Welding_Angle -20.0000,Welding_CDIS 5,Welding_ACC 100,Welding_Offset {X 0.0,Y 0.0,Z 0.0}}
L270_Welding_Craft[2,10]={Welding_Name[] "S10",Welding_Pos {X 533.000,Y 338.000,Z -2.05000,A 0.0,B -23.0000,C 0.0},Welding_Power 80.0000,Welding_Speed 0.0400000,Welding_Angle -20.0000,Welding_CDIS 5,Welding_ACC 100,Welding_Offset {X 0.0,Y 0.0,Z 0.0}}

DECL GLOBAL Surr_Welding_Craft_Type C315_Welding_Craft[2,3]
C315_Welding_Craft[1,1]={Welding_Name[] "C315_S1",Welding_Pos {X 366.000,Y 656.000,Z 0.0,A 0.0,B 0.0,C -20.0000},Welding_Power 80.0000,Welding_Speed 0.0400000,Welding_Angle -20.0000,Welding_CDIS 5,Welding_ACC 100,Welding_Offset {X 0.0,Y 0.0,Z 0.0}}
C315_Welding_Craft[1,2]={Welding_Name[] "PM3",Welding_Pos {X 373.071075,Y 653.071045,Z 0.0,A 0.0,B 0.0,C 0.0},Welding_Power 80.0000,Welding_Speed 0.0400000,Welding_Angle 20.0000,Welding_CDIS 5,Welding_ACC 100,Welding_Offset {X 0.0,Y 0.0,Z 0.0},Welding_Offset_CIR {C_X 0.0,C_Y 0.0,C_Z 0.0}}
C315_Welding_Craft[1,3]={Welding_Name[] "PE5",Welding_Pos {X 376.000,Y 646.000,Z 0.0,A 0.0,B 20.0000,C 0.0},Welding_Power 80.0000,Welding_Speed 0.0400000,Welding_Angle 20.0000,Welding_CDIS 5,Welding_ACC 100,Welding_Offset {X 0.0,Y 0.0,Z 0.0}}
C315_Welding_Craft[2,1]={Welding_Name[] "C315_S1",Welding_Pos {X 365.542,Y 725.577942,Z 0.0,A 0.0,B 0.0,C -20.0000},Welding_Power 80.0000,Welding_Speed 0.0300000,Welding_Angle -20.0000,Welding_CDIS 5,Welding_ACC 100,Welding_Offset {X 0.0,Y 0.0,Z 0.0}}
C315_Welding_Craft[2,2]={Welding_Name[] "PM7",Welding_Pos {X 371.833,Y 722.250,Z 0.0,A 0.0,B 0.0,C 0.0},Welding_Power 80.0000,Welding_Speed 0.0400000,Welding_Angle 20.0000,Welding_CDIS 5,Welding_ACC 100,Welding_Offset {X 0.0,Y 0.0,Z 0.0},Welding_Offset_CIR {C_X 0.0,C_Y 0.0,C_Z 0.0}}
C315_Welding_Craft[2,3]={Welding_Name[] "PE7",Welding_Pos {X 375.545074,Y 715.582,Z 0.0,A 0.0,B 20.0000,C 0.0},Welding_Power 80.0000,Welding_Speed 0.0150000,Welding_Angle 20.0000,Welding_CDIS 5,Welding_ACC 100,Welding_Offset {X -1.00000,Y 0.0,Z 0.0}}


DECL GLOBAL Surr_Welding_Craft_Type N45_Short_Craft[2,5]
N45_Short_Craft[1,1]={Welding_Name[] "S2",Welding_Pos {X 364.000,Y 0.0,Z -150.000,A 0.0,B 0.0,C 0.0},Welding_Power 80.0000,Welding_Speed 0.500000,Welding_Angle 0.0,Welding_CDIS 0,Welding_ACC 100,Welding_Offset {X 0.0,Y 0.0,Z 0.0}}
N45_Short_Craft[1,2]={Welding_Name[] "S13",Welding_Pos {X 364.000,Y 0.0,Z 0.0,A 0.0,B 0.0,C 0.0},Welding_Power 80.0000,Welding_Speed 0.500000,Welding_Angle 0.0,Welding_CDIS 0,Welding_ACC 100,Welding_Offset {X 0.0,Y 0.0,Z 0.0}}
N45_Short_Craft[1,3]={Welding_Name[] "S14",Welding_Pos {X 364.000,Y 23.0000,Z 0.0,A 0.0,B 0.0,C 0.0},Welding_Power 80.0000,Welding_Speed 0.01000000,Welding_Angle 0.0,Welding_CDIS 0,Welding_ACC 100,Welding_Offset {X 0.0,Y 0.0,Z 0.0}}
N45_Short_Craft[1,4]={Welding_Name[] "S4",Welding_Pos {X 364.000,Y 20.7000,Z -150.000,A 0.0,B 0.0,C 0.0},Welding_Power 80.0000,Welding_Speed 0.500000,Welding_Angle 0.0,Welding_CDIS 0,Welding_ACC 100,Welding_Offset {X 0.0,Y 0.0,Z 0.0}}
N45_Short_Craft[1,5]={Welding_Name[] "S12",Welding_Pos {X 28.9999981,Y 400.000,Z -3.00000,A 0.0,B 0.0,C -23.0000},Welding_Power 80.0000,Welding_Speed 0.500000,Welding_Angle 0.0,Welding_CDIS 0,Welding_ACC 100,Welding_Offset {X 0.0,Y 0.0,Z 0.0}}
N45_Short_Craft[2,1]={Welding_Name[] "S32",Welding_Pos {X 363.220,Y -0.316000,Z -150.000,A 0.0,B 0.0,C 0.0},Welding_Power 80.0000,Welding_Speed 0.500000,Welding_Angle 0.0,Welding_CDIS 0,Welding_ACC 100,Welding_Offset {X 0.0,Y 0.0,Z 0.0}}
N45_Short_Craft[2,2]={Welding_Name[] "S13",Welding_Pos {X 363.220,Y -0.316000,Z 0.0,A 0.0,B 0.0,C 0.0},Welding_Power 80.0000,Welding_Speed 0.500000,Welding_Angle 0.0,Welding_CDIS 0,Welding_ACC 100,Welding_Offset {X 0.0,Y 0.0,Z 0.0}}
N45_Short_Craft[2,3]={Welding_Name[] "S14",Welding_Pos {X 363.395,Y 19.3140,Z 0.0,A 0.0,B 0.0,C 0.0},Welding_Power 80.0000,Welding_Speed 0.01000000,Welding_Angle 0.0,Welding_CDIS 0,Welding_ACC 100,Welding_Offset {X 0.0,Y 0.0,Z 0.0}}
N45_Short_Craft[2,4]={Welding_Name[] "S4",Welding_Pos {X 363.323059,Y 11.2466183,Z -150.000,A 0.0,B 0.0,C 0.0},Welding_Power 80.0000,Welding_Speed 0.500000,Welding_Angle 0.0,Welding_CDIS 0,Welding_ACC 100,Welding_Offset {X 0.0,Y 0.0,Z 0.0}}
N45_Short_Craft[2,5]={Welding_Name[] "S12",Welding_Pos {X 28.9999981,Y 400.000,Z -3.00000,A 0.0,B 0.0,C -23.0000},Welding_Power 80.0000,Welding_Speed 0.500000,Welding_Angle 0.0,Welding_CDIS 0,Welding_ACC 100,Welding_Offset {X 0.0,Y 0.0,Z 0.0}}

DECL GLOBAL Surr_Welding_Craft_Type N135_Short_Craft[2,5]
N135_Short_Craft[1,1]={Welding_Name[] "S9",Welding_Pos {X 36.0000,Y 0.0,Z -150.000,A 0.0,B 0.0,C 0.0},Welding_Power 80.0000,Welding_Speed 0.500000,Welding_Angle 0.0,Welding_CDIS 0,Welding_ACC 100,Welding_Offset {X 0.0,Y 0.0,Z 0.0}}
N135_Short_Craft[1,2]={Welding_Name[] "S13",Welding_Pos {X 36.0000,Y 0.0,Z 0.0,A 0.0,B 0.0,C 0.0},Welding_Power 80.0000,Welding_Speed 0.500000,Welding_Angle 0.0,Welding_CDIS 0,Welding_ACC 100,Welding_Offset {X 0.0,Y 0.0,Z 0.0}}
N135_Short_Craft[1,3]={Welding_Name[] "S14",Welding_Pos {X 36.0000,Y 23.0000,Z 0.0,A 0.0,B 0.0,C 0.0},Welding_Power 80.0000,Welding_Speed 0.01000000,Welding_Angle 0.0,Welding_CDIS 0,Welding_ACC 100,Welding_Offset {X 0.0,Y 0.0,Z 0.0}}
N135_Short_Craft[1,4]={Welding_Name[] "S4",Welding_Pos {X 36.0000,Y 20.7000,Z -150.000,A 0.0,B 0.0,C 0.0},Welding_Power 80.0000,Welding_Speed 0.500000,Welding_Angle 0.0,Welding_CDIS 0,Welding_ACC 100,Welding_Offset {X 0.0,Y 0.0,Z 0.0}}
N135_Short_Craft[1,5]={Welding_Name[] "S12",Welding_Pos {X 28.9999981,Y 400.000,Z -3.00000,A 0.0,B 0.0,C -23.0000},Welding_Power 80.0000,Welding_Speed 0.500000,Welding_Angle 0.0,Welding_CDIS 0,Welding_ACC 100,Welding_Offset {X 0.0,Y 0.0,Z 0.0}}
N135_Short_Craft[2,1]={Welding_Name[] "S92",Welding_Pos {X 32.5260,Y -0.971000,Z -150.000,A 0.0,B 0.0,C 0.0},Welding_Power 80.0000,Welding_Speed 0.500000,Welding_Angle 0.0,Welding_CDIS 0,Welding_ACC 100,Welding_Offset {X 0.0,Y 0.0,Z 0.0}}
N135_Short_Craft[2,2]={Welding_Name[] "S13",Welding_Pos {X 32.5260,Y -0.971000,Z 0.0,A 0.0,B 0.0,C 0.0},Welding_Power 80.0000,Welding_Speed 0.500000,Welding_Angle 0.0,Welding_CDIS 0,Welding_ACC 100,Welding_Offset {X 0.0,Y 0.0,Z 0.0}}
N135_Short_Craft[2,3]={Welding_Name[] "S14",Welding_Pos {X 32.3940,Y 18.1940,Z 0.0,A 0.0,B 0.0,C 0.0},Welding_Power 80.0000,Welding_Speed 0.01000000,Welding_Angle 0.0,Welding_CDIS 0,Welding_ACC 100,Welding_Offset {X 0.0,Y 0.0,Z 0.0}}
N135_Short_Craft[2,4]={Welding_Name[] "S4",Welding_Pos {X 32.4600,Y 8.61150074,Z -150.000,A 0.0,B 0.0,C 0.0},Welding_Power 80.0000,Welding_Speed 0.500000,Welding_Angle 0.0,Welding_CDIS 0,Welding_ACC 100,Welding_Offset {X 0.0,Y 0.0,Z 0.0}}
N135_Short_Craft[2,5]={Welding_Name[] "S12",Welding_Pos {X 28.9999981,Y 400.000,Z -3.00000,A 0.0,B 0.0,C -23.0000},Welding_Power 80.0000,Welding_Speed 0.500000,Welding_Angle 0.0,Welding_CDIS 0,Welding_ACC 100,Welding_Offset {X 0.0,Y 0.0,Z 0.0}}

DECL GLOBAL Surr_Welding_Craft_Type N225_Short_Craft[2,5]
N225_Short_Craft[1,1]={Welding_Name[] "S10",Welding_Pos {X 36.0000,Y 680.000,Z -150.000,A 0.0,B 0.0,C 0.0},Welding_Power 80.0000,Welding_Speed 0.500000,Welding_Angle 0.0,Welding_CDIS 0,Welding_ACC 100,Welding_Offset {X 0.0,Y 0.0,Z 0.0}}
N225_Short_Craft[1,2]={Welding_Name[] "S13",Welding_Pos {X 36.0000,Y 680.000,Z 0.0,A 0.0,B 0.0,C 0.0},Welding_Power 80.0000,Welding_Speed 0.500000,Welding_Angle 0.0,Welding_CDIS 0,Welding_ACC 100,Welding_Offset {X 0.0,Y 0.0,Z 0.0}}
N225_Short_Craft[1,3]={Welding_Name[] "S14",Welding_Pos {X 36.0000,Y 657.000,Z 0.0,A 0.0,B 0.0,C 0.0},Welding_Power 80.0000,Welding_Speed 0.01000000,Welding_Angle 0.0,Welding_CDIS 0,Welding_ACC 100,Welding_Offset {X 0.0,Y 0.0,Z 0.0}}
N225_Short_Craft[1,4]={Welding_Name[] "S4",Welding_Pos {X 36.0000,Y 667.500,Z -150.000,A 0.0,B 0.0,C 0.0},Welding_Power 80.0000,Welding_Speed 0.500000,Welding_Angle 0.0,Welding_CDIS 0,Welding_ACC 100,Welding_Offset {X 0.0,Y 0.0,Z 0.0}}
N225_Short_Craft[1,5]={Welding_Name[] "S12",Welding_Pos {X 28.9999981,Y 400.000,Z -3.00000,A 0.0,B 0.0,C -23.0000},Welding_Power 80.0000,Welding_Speed 0.500000,Welding_Angle 0.0,Welding_CDIS 0,Welding_ACC 100,Welding_Offset {X 0.0,Y 0.0,Z 0.0}}
N225_Short_Craft[2,1]={Welding_Name[] "S13",Welding_Pos {X 31.6330,Y 679.439,Z -150.000,A 0.0,B 0.0,C 0.0},Welding_Power 80.0000,Welding_Speed 0.500000,Welding_Angle 0.0,Welding_CDIS 0,Welding_ACC 100,Welding_Offset {X 0.0,Y 0.0,Z 0.0}}
N225_Short_Craft[2,2]={Welding_Name[] "S13",Welding_Pos {X 31.6330,Y 679.439,Z 0.0,A 0.0,B 0.0,C 0.0},Welding_Power 80.0000,Welding_Speed 0.500000,Welding_Angle 0.0,Welding_CDIS 0,Welding_ACC 100,Welding_Offset {X 0.0,Y 0.0,Z 0.0}}
N225_Short_Craft[2,3]={Welding_Name[] "S14",Welding_Pos {X 31.8670,Y 660.025,Z 0.0,A 0.0,B 0.0,C 0.0},Welding_Power 80.0000,Welding_Speed 0.01000000,Welding_Angle 0.0,Welding_CDIS 0,Welding_ACC 100,Welding_Offset {X 0.0,Y 0.0,Z 0.0}}
N225_Short_Craft[2,4]={Welding_Name[] "S4",Welding_Pos {X 31.7500,Y 669.732056,Z -150.000,A 0.0,B 0.0,C 0.0},Welding_Power 80.0000,Welding_Speed 0.500000,Welding_Angle 0.0,Welding_CDIS 0,Welding_ACC 100,Welding_Offset {X 0.0,Y 0.0,Z 0.0}}
N225_Short_Craft[2,5]={Welding_Name[] "S12",Welding_Pos {X 28.9999981,Y 400.000,Z -3.00000,A 0.0,B 0.0,C -23.0000},Welding_Power 80.0000,Welding_Speed 0.500000,Welding_Angle 0.0,Welding_CDIS 0,Welding_ACC 100,Welding_Offset {X 0.0,Y 0.0,Z 0.0}}

DECL GLOBAL Surr_Welding_Craft_Type N315_Short_Craft[2,5]
N315_Short_Craft[1,1]={Welding_Name[] "S17",Welding_Pos {X 364.000,Y 680.000,Z -150.000,A 0.0,B 0.0,C 0.0},Welding_Power 80.0000,Welding_Speed 0.500000,Welding_Angle 0.0,Welding_CDIS 0,Welding_ACC 100,Welding_Offset {X 0.0,Y 0.0,Z 0.0}}
N315_Short_Craft[1,2]={Welding_Name[] "S13",Welding_Pos {X 364.000,Y 680.000,Z 0.0,A 0.0,B 0.0,C 0.0},Welding_Power 80.0000,Welding_Speed 0.500000,Welding_Angle 0.0,Welding_CDIS 0,Welding_ACC 100,Welding_Offset {X 0.0,Y 0.0,Z 0.0}}
N315_Short_Craft[1,3]={Welding_Name[] "S14",Welding_Pos {X 364.000,Y 657.000,Z 0.0,A 0.0,B 0.0,C 0.0},Welding_Power 80.0000,Welding_Speed 0.01000000,Welding_Angle 0.0,Welding_CDIS 0,Welding_ACC 100,Welding_Offset {X 0.0,Y 0.0,Z 0.0}}
N315_Short_Craft[1,4]={Welding_Name[] "S4",Welding_Pos {X 364.000,Y 667.500,Z -150.000,A 0.0,B 0.0,C 0.0},Welding_Power 80.0000,Welding_Speed 0.500000,Welding_Angle 0.0,Welding_CDIS 0,Welding_ACC 100,Welding_Offset {X 0.0,Y 0.0,Z 0.0}}
N315_Short_Craft[1,5]={Welding_Name[] "S12",Welding_Pos {X 28.9999981,Y 400.000,Z -3.00000,A 0.0,B 0.0,C -23.0000},Welding_Power 80.0000,Welding_Speed 0.500000,Welding_Angle 0.0,Welding_CDIS 0,Welding_ACC 100,Welding_Offset {X 0.0,Y 0.0,Z 0.0}}
N315_Short_Craft[2,1]={Welding_Name[] "S17",Welding_Pos {X 362.986,Y 679.910,Z -150.000,A 0.0,B 0.0,C 0.0},Welding_Power 80.0000,Welding_Speed 0.500000,Welding_Angle 0.0,Welding_CDIS 0,Welding_ACC 100,Welding_Offset {X 0.0,Y 0.0,Z 0.0}}
N315_Short_Craft[2,2]={Welding_Name[] "S13",Welding_Pos {X 362.986,Y 679.910,Z 0.0,A 0.0,B 0.0,C 0.0},Welding_Power 80.0000,Welding_Speed 0.500000,Welding_Angle 0.0,Welding_CDIS 0,Welding_ACC 100,Welding_Offset {X 0.0,Y 0.0,Z 0.0}}
N315_Short_Craft[2,3]={Welding_Name[] "S14",Welding_Pos {X 363.044,Y 660.468,Z 0.0,A 0.0,B 0.0,C 0.0},Welding_Power 80.0000,Welding_Speed 0.01000000,Welding_Angle 0.0,Welding_CDIS 0,Welding_ACC 100,Welding_Offset {X 0.0,Y 0.0,Z 0.0}}
N315_Short_Craft[2,4]={Welding_Name[] "S4",Welding_Pos {X 363.015,Y 670.188965,Z -150.000,A 0.0,B 0.0,C 0.0},Welding_Power 80.0000,Welding_Speed 0.500000,Welding_Angle 0.0,Welding_CDIS 0,Welding_ACC 100,Welding_Offset {X 0.0,Y 0.0,Z 0.0}}
N315_Short_Craft[2,5]={Welding_Name[] "S12",Welding_Pos {X 28.9999981,Y 400.000,Z -3.00000,A 0.0,B 0.0,C -23.0000},Welding_Power 80.0000,Welding_Speed 0.500000,Welding_Angle 0.0,Welding_CDIS 0,Welding_ACC 100,Welding_Offset {X 0.0,Y 0.0,Z 0.0}}



DECL GLOBAL Surround_Welding_Type N1_Sink_Data={Sink_Size_Long 632.000,Sink_Size_Width 347.000,Sink_Size_R 12.0000,Sink_Size_Short_Side 23.0000,Sink_Size_Short_OnePos 36.0000,Sink_Size_Short_TwoPos 323.000,Sink_Size_Pots_Thick 0.0,Sink_Size_Panel_Thick 0.0,Sink_Model 952128,Sink_Size_Left_Distance 24.0000,Sink_Size_Down_Distance 24.0000,Sink_Type #LeftRight_One}
DECL GLOBAL Surround_Welding_Type N2_Sink_Data={Sink_Size_Long 700.000,Sink_Size_Width 350.000,Sink_Size_R 10.0000,Sink_Size_Short_Side 23.0000,Sink_Size_Short_OnePos 36.0000,Sink_Size_Short_TwoPos 328.000,Sink_Size_Pots_Thick 0.0,Sink_Size_Panel_Thick 0.0,Sink_Model 952212,Sink_Size_Left_Distance 25.0000,Sink_Size_Down_Distance 25.0000,Sink_Type #LeftRight_One}
;-----------Viion_INI------------



DECL GLOBAL INT Vision_Scope=20
;GLOBAL CHAR $Socket_Connect[1024]
;DECL GLOBAL CHAR $SOCKET_MESS[1024]
;DECL GLOBAL MODEL_TYPE $N_1
;DECL GLOBAL MODEL_TYPE $N_2
;DECL GLOBAL INT $MY_Work_Number=-1



;----------------------------------
ENDDAT
